FUNCTION_BLOCK SK_MoveNeedleDown (* Lower the needle to Distance mm below the top; the default is all the way down (parameters: Distance [mm] 0.0..50.0, default 50.0). START -> SUCCESS or FAILURE; OPC UA SetParameters(Session, ...) -> [Accepted, ErrorID]; parameter inputs are the instance's defaults *)
  (* Standard: 61499-2 *)
  (* Version 0.1, 2026-09-28, Project contributors, AAU Smart Production Lab *)
  PACKAGE filler;
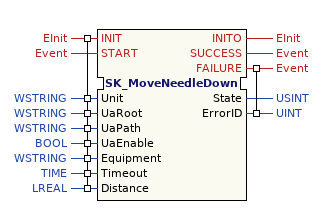
  EVENT_INPUT
    INIT : EInit WITH Unit, UaRoot, UaPath, UaEnable, Equipment, Timeout, Distance;
    START;
  END_EVENT
  EVENT_OUTPUT
    INITO : EInit;
    SUCCESS;
    FAILURE WITH ErrorID;
  END_EVENT
  VAR_INPUT
    Unit : WSTRING;
    UaRoot : WSTRING;
    UaPath : WSTRING;
    UaEnable : BOOL;
    Equipment : WSTRING := "NeedleAxis";
    Timeout : TIME := T#5s;
    Distance : LREAL := 50.0;
  END_VAR
  VAR_OUTPUT
    State : USINT;
    ErrorID : UINT;
  END_VAR
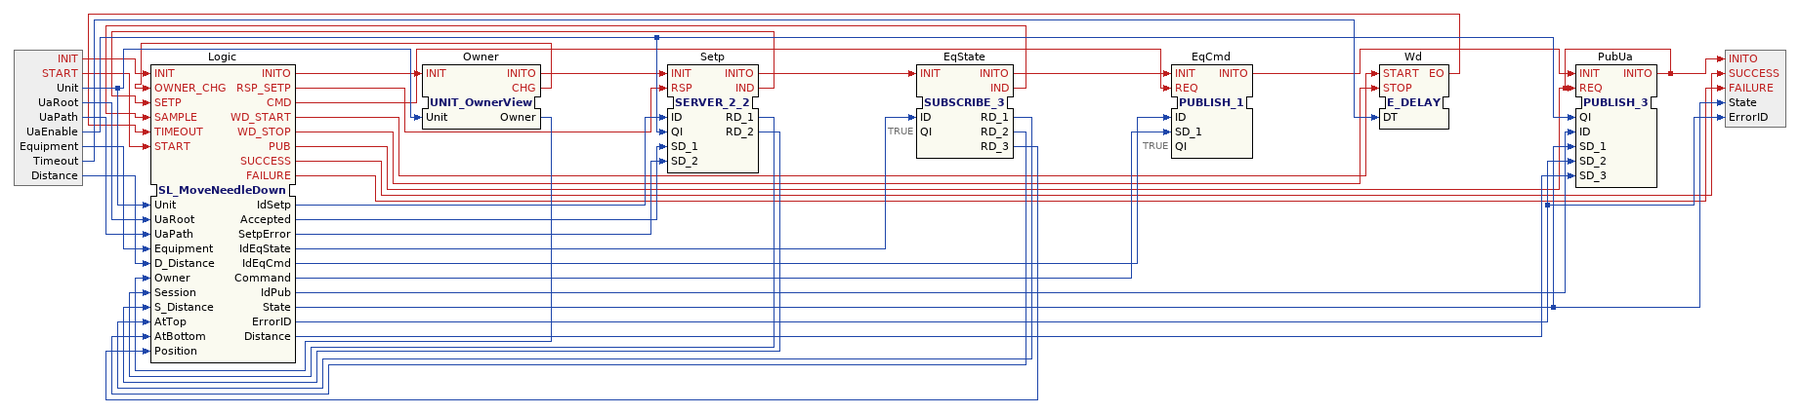
  FBS
    Logic : filler::SL_MoveNeedleDown;
    Owner : unitlib::UNIT_OwnerView;
    Setp : iec61499::net::SERVER_2_2;
    EqState : iec61499::net::SUBSCRIBE_3(QI := TRUE);
    EqCmd : iec61499::net::PUBLISH_1(QI := TRUE);
    Wd : iec61499::events::E_DELAY;
    PubUa : iec61499::net::PUBLISH_3;
  END_FBS
  EVENT_CONNECTIONS
    INIT TO Logic.INIT;
    Logic.INITO TO Owner.INIT;
    Owner.INITO TO Setp.INIT;
    Setp.INITO TO EqState.INIT;
    EqState.INITO TO EqCmd.INIT;
    EqCmd.INITO TO PubUa.INIT;
    PubUa.INITO TO PubUa.REQ;
    PubUa.INITO TO INITO;
    Owner.CHG TO Logic.OWNER_CHG;
    Setp.IND TO Logic.SETP;
    Logic.RSP_SETP TO Setp.RSP;
    EqState.IND TO Logic.SAMPLE;
    Logic.CMD TO EqCmd.REQ;
    Logic.WD_START TO Wd.START;
    Logic.WD_STOP TO Wd.STOP;
    Wd.EO TO Logic.TIMEOUT;
    Logic.PUB TO PubUa.REQ;
    START TO Logic.START;
    Logic.SUCCESS TO SUCCESS;
    Logic.FAILURE TO FAILURE;
  END_CONNECTIONS
  DATA_CONNECTIONS
    Unit TO Logic.Unit;
    UaRoot TO Logic.UaRoot;
    UaPath TO Logic.UaPath;
    Equipment TO Logic.Equipment;
    Distance TO Logic.D_Distance;
    Unit TO Owner.Unit;
    Owner.Owner TO Logic.Owner;
    Logic.IdSetp TO Setp.ID;
    UaEnable TO Setp.QI;
    UaEnable TO PubUa.QI;
    Setp.RD_1 TO Logic.Session;
    Setp.RD_2 TO Logic.S_Distance;
    Logic.Accepted TO Setp.SD_1;
    Logic.SetpError TO Setp.SD_2;
    Logic.IdEqState TO EqState.ID;
    EqState.RD_1 TO Logic.AtTop;
    EqState.RD_2 TO Logic.AtBottom;
    EqState.RD_3 TO Logic.Position;
    Logic.IdEqCmd TO EqCmd.ID;
    Logic.Command TO EqCmd.SD_1;
    Timeout TO Wd.DT;
    Logic.IdPub TO PubUa.ID;
    Logic.State TO PubUa.SD_1;
    Logic.State TO State;
    Logic.ErrorID TO PubUa.SD_2;
    Logic.ErrorID TO ErrorID;
    Logic.Distance TO PubUa.SD_3;
  END_CONNECTIONS
END_FUNCTION_BLOCK
